// TIA Portal V17 export
// export: Created 2025-03-07T09:23:46.5137202Z, ExportSetting WithDefaults, DisplayName Totally Integrated Automation Portal, DisplayVersion V17 Update 8, DisplayName TIA Portal Openness, DisplayVersion V17 Update 8, DisplayName TIA Portal Version Control Interface, DisplayVersion V17, DisplayName SINAMICS Startdrive Advanced, DisplayVersion V17 SP2, DisplayName SINAMICS Startdrive G110M, G120, G120C, G120D, G120P, G115D, DisplayVersion V17 SP2, DisplayName SINAMICS Startdrive G130, G150, S120, S150, SINAMICS MV, S210, DisplayVersion V17 SP2, DisplayName STEP 7 Professional, DisplayVersion V17 Update 8, DisplayName SINUMERIK ONE STEP 7 Toolbox, DisplayVersion V17 Update 12, DisplayName SINUMERIK 840D sl STEP 7 Toolbox, DisplayVersion V17 Update 12, DisplayName STEP 7 Safety, DisplayVersion V17 Update 6, DisplayName WinCC Advanced, DisplayVersion V17 Update 8
DATA_BLOCK "DB7260_PLC_HMI_GENERAL"   // DB7260
{ DB_Accessible_From_OPC_UA := 'FALSE' }
VERSION : 0.1
// stored: AutoNumber false, DBAccessibleFromOPCUA false, DBAccessibleFromWebserver true, InstanceOfName FB7239_VARIABLES_PLC_HMI_GENERAL, InstanceOfType FB
"FB7239_VARIABLES_PLC_HMI_GENERAL"
   // VAR_INPUT
   //    FEEDERS_MANUAL_MODE : Bool;
   //    FEEDERS_AUTO_MODE : Bool;
   //    HOPPERS_MANUAL_MODE : Bool;
   //    HOPPERS_AUTO_MODE : Bool;
   // END_VAR
   // VAR_OUTPUT
   //    FEEDERS_MODE_STATE : Int;
   //    HOPPERS_MODE_STATE : Int;
   // END_VAR
BEGIN
END_DATA_BLOCK
